(* CoDeSys 2.3.9.59 project: Pistone SFC.pro *)
(* Libraries: Iecsfc.lib 12.5.98 12:03:00, STANDARD.LIB *)

(* Task configuration *)
TASK Standard (PRIORITY := 0, INTERVAL := T#10ms);
	MAIN
END_TASK

(* POU MAIN, SFC *)
PROGRAM MAIN
VAR
(*Variabili Pistone*)
         (*Ingressi*)
	pezzo_magazzino  AT%IX0.0:BOOL;
	pistone_avanti AT%IX0.2:BOOL;
	pistone_indietro AT%IX0.4:BOOL;
         pulsante: BOOL;
         (*Uscite*)
	pistone_on  AT%QX0.2:BOOL;

(*Variabili Nastro*)
         (*Ingressi*)
	fine_corsa_nastro  AT%IX0.6:BOOL;
         (*Uscite*)
	nastro_on  AT%QX0.0:BOOL;

END_VAR
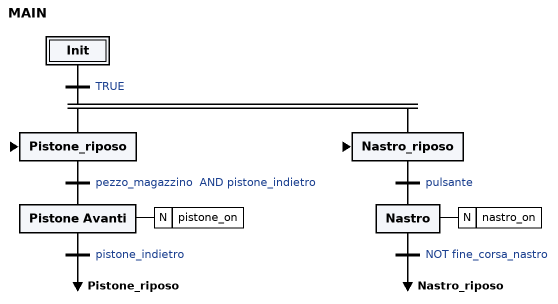
INITIAL_STEP Init:
END_STEP
TRANSITION FROM Init TO (Pistone_riposo, Nastro_riposo) := TRUE;
END_TRANSITION
STEP Pistone_riposo:
END_STEP
TRANSITION FROM Pistone_riposo TO Pistone Avanti := pezzo_magazzino  AND pistone_indietro;
END_TRANSITION
STEP Nastro_riposo:
END_STEP
TRANSITION FROM Nastro_riposo TO Nastro  := pulsante;
END_TRANSITION
STEP Nastro :
	nastro_on(N);
END_STEP
TRANSITION FROM Nastro  TO Nastro_riposo := NOT fine_corsa_nastro;
END_TRANSITION
STEP Pistone Avanti:
	pistone_on(N);
END_STEP
TRANSITION FROM Pistone Avanti TO Pistone_riposo := pistone_indietro;
END_TRANSITION
END_PROGRAM

(* Visualisation Pulsante
ellipse at (140,80)-(271,211): text "Pulsante"; toggles MAIN.pulsante
*)
